{attribute 'pack_mode' := '1'} 
TYPE ASCF_CC_OPCUACS_Reader_Temp_Bool :
STRUCT
	stReadListReturnInfo	: ARRAY [1..2] OF ST_UAReadListReturnInfo;
	QC		: BYTE	:= 16#0;
	Value	: BOOL	:= FALSE;
END_STRUCT
END_TYPE

(* stored: Version 1.1.0.1, ProductVersion 3.1.4026.4
   DUT ASCF_CC_OPCUACS_Reader_Temp_Bool: Id {3a99807b-d748-4cb8-9261-b0f9ae026d74} *)
